Yaskawa INFORM job: WELDGAS.JBI

/JOB
//NAME WELDGAS
//POS
///NPOS 0,0,0,0,0,0
//INST
///DATE 2015/09/29 09:04
///ATTR SC,RW,MC
NOP
DOUT OT#(18) OFF
TIMER T=0.50
DOUT OT#(19) ON
END
